RoboDK station: Yuchen_2024.rdk

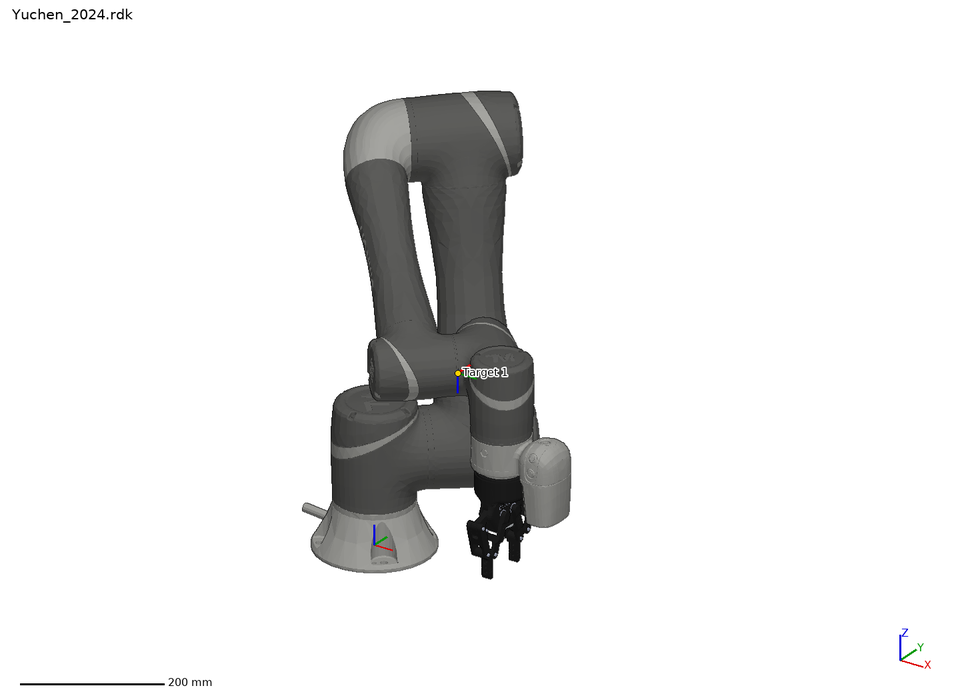
[picture v0: the station drawn from its stored meshes, robots at their saved joint values, targets as dots, program paths as lines]
Station Yuchen_2023 (saved by RoboDK 5.5.3). Poses are relative to the parent item; angles as X-Y-Z fixed-axis rotations.
  - frame Omron TM5-900 Base at (0, 0, 0) mm
    - robot Omron TM5-900: 6 axes, payload 4 kg, reach 900 mm, repeatability 0.1 mm, weight 30 kg
        modified DH rows (alpha deg, a mm, theta deg, d mm): 0, 0, 0, 145.2; 90, 0, 90, 0; 0, 429, 0, 0; 0, 411, -90, 122.3; -90, 0, 0, 106.5; 90, 0, 180, 114.15
        joint limits [-270, -180, -155, -180, -180, -270] to [270, 180, 155, 180, 180, 270]; home [0, 0, 90, -90, 90, 0]; saved at [134.48, 19.77, -133.5, 23.17, -90.14, -45.91]
      - tool RobotiQ 2F-85 Gripper (Closed), TCP at (0, 0, 130) mm, size 134.4 x 75 x 157.6 mm
    - frame Frame 2 at (241, -142.19, 389.18) mm, rotated rx -179.52 ry -0.29 rz 90.39 deg
      - target Target 1 (Cartesian target) at (0, 0, 0) mm; joints [123.542, 38.198, -125.271, -2.927, -90, -56.458] of Omron TM5-900
  - Python program Reading_CaseStudy (listed below)
  - Python program 20240725_OPT (listed below)

--- Python program Reading_CaseStudy ---
# PS C:\Users\Tesisti> python -m venv hrcreading
# PS C:\Users\Tesisti> .\hrcreading\Scripts\activate
# (hrcreading) PS C:\Users\Tesisti> C:/Python310/python.exe c:/Users/Tesisti/AppData/Local/Temp/Reading_CaseStudy_3.py

# import os
# os.environ['OPENAI_API_KEY'] ='sk-proj-5TX9ug0B6qDGBHHPTzqzT3BlbkFJDqqZnPh7HjYkSIwuRGDw'

# sys.path.append(yolov7_path)
# print("sys.path:", sys.path)
import cv2
import torch
import pyttsx3
from datetime import datetime
import numpy as np
import requests
from IPython.display import display, Audio
import openai
import time
from PIL import Image, ImageTk
import pandas as pd
import matplotlib.pyplot as plt
import pygame
import os
from GUI import AssemblyGUI
import tkinter as tk
from playsound import playsound
import sys
import tkinter as tk
from tkinter import ttk, messagebox
import pygame
from PIL import Image, ImageTk
from playsound import playsound


# from ultralytics.yolo.utils.downloads import non_max_suppression, check_img_size, scale_coords
# from utils.general import non_max_suppression, check_img_size, scale_coords
# from utils.torch_utils import select_device



# ———————————————————————————————————————————————————————————— GUI design ————————————————————————————————————————————————————————————
def load_and_play(speech=None):
    try:
        playsound(speech)
    except Exception as e:
        print(f"Error playing {speech}: {e}")

def pause_audio():
    pygame.mixer.music.pause()

def set_volume(value):
    volume_level = float(value) / 100
    pygame.mixer.music.set_volume(volume_level)

def change_voice(selected_voice_type):
    voice_type = selected_voice_type
    load_and_play()

def create_gui():
    root.title("Assembly Monitoring System")
    root.geometry("1200x800")  # Adjust window size

    # Frames for different sections
    left_column = tk.Frame(self.root, width=800, bg='white')
    right_column = tk.Frame(self.root, width=400, bg='light gray')
    left_column.pack(side='left', fill='both', expand=True)
    right_column.pack(side='right', fill='both', expand=True)

    # Sub-frames within the left frame
    image_display_frame = tk.Frame(left_column, width=800)
    label_description_0 = tk.Label(image_display_frame, text="Multi-form Instructions", font=('Arial', 16, 'bold'))
    label_description_0.pack(pady=(20, 0))
    image_display_frame.pack(side="top", fill="both", expand=True)
    command_frame = tk.Frame(left_column, width=400)
    command_frame.pack(side="top", fill="both", expand=False)

    # Sub-frames for each image and its description
    left_image_frame = tk.Frame(image_display_frame, width=400)
    right_image_frame = tk.Frame(image_display_frame, width=400)
    left_image_frame.pack(side="left", fill="both", expand=True)
    right_image_frame.pack(side="right", fill="both", expand=True)

    # Labels and images in the left image frame
    label_description_1 = tk.Label(left_image_frame, text="Component", font=('Arial', 14))
    canvas_com = tk.Canvas(left_image_frame, bg="gray", height=80, width=80)
    label_operation_1 = tk.Label(left_image_frame, text="Operation", font=('Arial', 14))
    canvas_ope = tk.Canvas(left_image_frame, bg="gray", height=80, width=80)
    label_description_1.pack(pady=(20, 0))
    canvas_com.pack(pady=(5, 5), fill="both", expand=True)
    label_operation_1.pack(pady=(5, 0))
    canvas_ope.pack(pady=(5, 20), fill="both", expand=True)

    # Labels and images in the right image frame
    label_description_2 = tk.Label(right_image_frame, text="Tool", font=('Arial', 14))
    canvas_too = tk.Canvas(right_image_frame, bg="gray", height=80, width=80)
    label_operation_2 = tk.Label(right_image_frame, text="Assembly Result", font=('Arial', 14))
    canvas_res = tk.Canvas(right_image_frame, bg="gray", height=80, width=80)
    label_description_2.pack(pady=(20, 0))
    canvas_too.pack(pady=(5, 5), fill="both", expand=True)
    label_operation_2.pack(pady=(5, 0))
    canvas_res.pack(pady=(5, 20), fill="both", expand=True)

    # Text box for instructions
    text_frame = tk.Frame(left_column, width=400)
    text_frame.pack(side="top", fill="both", expand=False, pady=(0, 0))
    text_instruction = tk.Text(text_frame, height=10, width=80)
    text_instruction.pack(pady=(5, 5), padx=0)

    # Main command frame for holding all control elements
    command_frame = tk.Frame(left_column, bg='white')
    command_frame.pack(fill="x")

    # Controls frame for holding buttons and sliders horizontally
    controls_frame = tk.Frame(command_frame)
    controls_frame.pack(fill="x", expand=True)

    # Buttons and controls in the command frame
    play_button = tk.Button(controls_frame, text="Play Instructions", font=('Arial', 12), command=load_and_play(speech=None))
    pause_button = tk.Button(controls_frame, text="Pause Instructions", font=('Arial', 12), command=pause_audio())
    volume_control = tk.Scale(controls_frame, from_=0, to=100, orient="horizontal", label="Volume", font=('Arial', 12), command=set_volume)
    volume_control.set(50)  # Default volume set to 50%
    sound_type = ttk.Combobox(controls_frame, values=["Male", "Female"], font=('Arial', 12), state="readonly")
    sound_type.set("Male")  # Default sound type
    play_button.grid(row=0, column=0, padx=10, pady=10, sticky="ew")
    pause_button.grid(row=0, column=1, padx=10, pady=10, sticky="ew")
    volume_control.grid(row=0, column=2, padx=10, pady=10, sticky="ew")
    sound_type.grid(row=0, column=3, padx=10, pady=10, sticky="ew")

    # Right column single image frame
    realtime_image_frame = tk.Frame(right_column, width=400, bg='light blue')
    realtime_image_frame.pack(side="top", fill="both", expand=True)
    label_description_3 = tk.Label(realtime_image_frame, text="Actual Statu", font=('Arial', 16, 'bold'), bg='light blue')
    label_description_3.pack(pady=(20, 0))

    # Image and label in the right column
    label_description_realtime = tk.Label(realtime_image_frame, text="Real-time Image", font=('Arial', 14), bg='light blue')
    realtime_canvas = tk.Canvas(realtime_image_frame, bg="gray", height=300, width=450)
    label_description_realtime.pack(pady=(20, 0))
    realtime_canvas.pack(pady=(5, 5), fill="none", expand=False)

    # Text box for assembly progress
    progress_frame = tk.Frame(right_column, width=400, bg='light blue')
    progress_frame.pack(side="top", fill="both", expand=False, pady=(0, 0))
    progress_label = tk.Label(progress_frame, text="Assembly Status", font=('Arial', 14), bg='light blue')
    progress_label.pack()
    progress_text = tk.Text(progress_frame, height=15, width=56)
    progress_text.pack(pady=(5, 20), padx=20)

    # Button frame at the bottom of right_column
    button_frame = tk.Frame(right_column, bg='light blue')
    button_frame.pack(side='bottom', fill='x', expand=False)
    exit_button = tk.Button(button_frame, text="Exit", font=('Arial', 12), command=root.destroy, width=10)
    error_button = tk.Button(button_frame, text="Report Error", font=('Arial', 12), command=lambda: messagebox.showerror("Error", "System Error Reported"), width=20)
    exit_button.pack(side="left", padx=35, pady=25)
    error_button.pack(side="right", padx=35, pady=25)




# ———————————————————————————————————————————————————————————— Data and model Setting ————————————————————————————————————————————————————————————
# YOLOv7
# loading the pre-trained YOLOv7 model
yolov7_path = 'C:/Users/Tesisti/Desktop/Yuchen 2023-2026/06 GPT+YOLOV7/yolov7'
weights_path = 'C:/Users/Tesisti/Desktop/Yuchen 2023-2026/06 GPT+YOLOV7/yolov7/best.pt'
device = torch.device('cuda' if torch.cuda.is_available() else 'cpu')
model = torch.hub.load(yolov7_path, 'custom', weights_path, source='local').to(device)
model.eval() # 确保模型处于评估模式
yolov7_label_order = ['Allen key', 'Hex cap screw (big)', 'Drive shaft companion flange', 'Nuts', 'Pump housing', 'S12', 'S6', 'S9', 'Washers', 'Wrench size 13']

# Assembly data loading
assembly_tasks_path = 'C:/Users/Tesisti/Desktop/Yuchen 2023-2026/06 GPT+YOLOV7/assembly_tasks.xlsx'
assembly_tasks_df = pd.read_excel(assembly_tasks_path)
index_total = assembly_tasks_df.dropna(how='all').shape[0] - 1

steps_classes = assembly_tasks_df['step'].dropna().to_dict()
components_classes = assembly_tasks_df['components'].dropna().to_dict()
tools_classes = assembly_tasks_df['tools'].dropna().to_dict()
operations_classes = assembly_tasks_df['operations'].dropna().to_dict()
time_classes = assembly_tasks_df['time'].dropna().to_dict()
lastorder_classes = assembly_tasks_df['lastorder'].dropna().to_dict()
print(steps_classes)
print(components_classes)
print(tools_classes)

# Error information
error_templates_path = 'C:/Users/Tesisti/Desktop/Yuchen 2023-2026/06 GPT+YOLOV7/error_templates.xlsx'
error_templates_df = pd.read_excel(error_templates_path)
error_templates = dict(zip(error_templates_df['error_type'], error_templates_df['template']))
print(error_templates)



# ———————————————————————————————————————————————————————————— Image Capture and Process ————————————————————————————————————————————————————————————
# Image display
def show_image(frame):
    try:
        frame_rgb = cv2.cvtColor(frame, cv2.COLOR_BGR2RGB)
        plt.imshow(frame_rgb)
        plt.axis('off')
        timestamp = datetime.now().strftime("%Y%m%d%H%M%S")
        plt.title(f'Image_{timestamp}')
        plt.show()  # Ensure the image is displayed when the function is called
    except Exception as e:
        print(f"Failed to display image: {e}")

# Image preprocessing
def preprocess_image(frame):
    try:
        img = cv2.cvtColor(frame, cv2.COLOR_BGR2RGB)
        img = img.astype(np.float32) / 255.0
        img = np.transpose(img, (2, 0, 1))
        img = np.expand_dims(img, 0)
        img = torch.from_numpy(img).float()
        return img
    except Exception as e:
        print(f"Error during image preprocessing: {e}")
        return None

# Image preprocessing cancel
def postprocess_image(tensor):
    if isinstance(tensor, torch.Tensor):
        tensor = tensor.cpu()
        image_np = tensor.numpy()
        image_np = image_np[0]
        if image_np.shape[0] < image_np.shape[2]:
            image_np = image_np.transpose(1, 2, 0)
        if image_np.max() <= 1.0:
            image_np = (image_np * 255).astype(np.uint8)
        return image_np
    else:
        print("传入的数据不是 torch.Tensor 类型")
        return None

# Image capturing
def capture_image():
    cap = cv2.VideoCapture(0)
    ret, frame = cap.read()
    cap.release()
    if ret:
        # show_image(frame)
        img = preprocess_image(frame)
        return img
    else:
        return None


# ———————————————————————————————————————————————————————————— YOLOv7 Detection and classification ————————————————————————————————————————————————————————————
# Image YOLOv7 detection
def detect_items(image):
    frame = image.squeeze().numpy().transpose(1, 2, 0) * 255  # 转换图像为适合显示的格式
    frame = frame.astype(np.uint8)

    with torch.no_grad():
        predictions = model(image)  # 使用模型进行预测
        predictions = predictions[0] if isinstance(predictions, tuple) else predictions
        predictions = non_max_suppression(predictions, conf_thres=0.6, iou_thres=0.45)

    detected_items = []  # 初始化检测到的物体列表

    # 检查predictions是否存在且不为空
    if predictions is not None and len(predictions) > 0 and len(predictions[0]) > 0:
        detected_items = predictions[0]  # 提取检测到的物体
        print(f"YOLOv7 detections found: {len(detected_items)}")  # 打印检测到的物体数量
    else:
        print("No detections found.")

    return detected_items

# detected items classification
def classify_detections(detected):
    classified_items = {
        'components': [],
        'tools': [],
        'steps': []
    }
    for detection in detected:
        x1, y1, x2, y2, conf, cls = detection[:6]
        if conf > 0.5:
            label = yolov7_label_order[int(cls)]
            print('label:' + label)
            if any(label == step for step in steps_classes.values()):
                classified_items['steps'].append(label)
            if any(label in component for component in components_classes.values()):
                classified_items['components'].append(label)
            if any(label in tool for tool in tools_classes.values()):
                classified_items['tools'].append(label)
    return classified_items



# ———————————————————————————————————————————————————————————— Annotate by Error ————————————————————————————————————————————————————————————
# Error validation and handle
def error_validation(classified, step_details, operator_name, location, item_type, task):
    details = {
        'now': datetime.now().strftime("%Y-%m-%d %H:%M"),
        'operator_name': operator_name,
        'location': location,
        'expected': step_details[item_type],
        'actual': classified[item_type],
        'step': step_details['step'],
        'task': task
    }

    error_result = {
        'type': item_type,
        'specific': details['actual'],
        'result': True
    }

    if set(details['actual']).issubset(set(details['expected'])):
        error_result['result'] = True
        error_log = None
    else:
        error_result['result'] = False
        error_log = error_templates[item_type].format(**details)  # Ensure error_templates is defined with proper templates.

    errorLog_dir = "C:/Users/Tesisti/Desktop/Yuchen 2023-2026/06 GPT+YOLOV7/Results_ErrorLog"
    current_time = datetime.now().strftime("%Y-%m-%d_%H-%M-%S")
    errorLog_filename = f"{errorLog_dir}/text{current_time}.txt"
    with open(errorLog_filename, "w") as text_file:
        text_file.write(error_log)
    print(f"Error log saved.")

    return error_result, error_log

# Label with different colors according to different situation
def annotate_image_with_labels(image, detected_items, classified_items, item_type, error_result):
    # Define colors for different scenarios
    correct_color = (0, 255, 0)  # Green for "True"
    wrong_color = (255, 0, 0)    # Red for "False"
    neutral_color = (128, 128, 128)  # Gray for other categories

    # Process the image once
    processed_image = postprocess_image(image)

    for detection in detected_items:
        x1, y1, x2, y2, conf, cls = detection[:6]
        detection_label = yolov7_label_order[int(cls)]  # Convert class ID to readable label

        # Determine the color based on classification and result
        if detection_label in classified_items[item_type]:
            color = correct_color if error_result['result'] else wrong_color
        else:
            color = neutral_color

        # Draw rectangle and label on the same processed image
        cv2.rectangle(processed_image, (int(x1), int(y1)), (int(x2), int(y2)), color, 2)
        cv2.putText(processed_image, detection_label, (int(x1), int(y1) - 10), cv2.FONT_HERSHEY_SIMPLEX, 0.5, color, 2)

    # Save and optionally display the annotated image
    timestamp = datetime.now().strftime("%Y%m%d%H%M%S")
    annotated_image_path = f'./Results_Image/annotated_{item_type}_{timestamp}.jpg'
    cv2.imwrite(annotated_image_path, processed_image)
    print(f"Annotated image saved.")

    return processed_image



# ———————————————————————————————————————————————————————————— GPT promt and speech ————————————————————————————————————————————————————————————
# Load gpt prompt
def generate_prompt(step_details, error_description):
    gpt_prompt_path = 'C:/Users/Tesisti/Desktop/Yuchen 2023-2026/06 GPT+YOLOV7/gpt_prompt.xlsx'
    gpt_prompt_df = pd.read_excel(gpt_prompt_path)
    prompt_template = gpt_prompt_df['prompt'].iloc[0]
    prompt = prompt_template.format(step_details=step_details, error_description=error_description)
    return prompt

def GPT_TTS(prompt):
    # Check GPT API key
    api_key = os.getenv('OPENAI_API_KEY')
    if not api_key:
        raise ValueError("API key is not set. Please ensure the 'OPENAI_API_KEY' environment variable is defined.")

    # Step1: Text generation
    response = openai.chat.completions.create(
        model="gpt-4o",
        messages=[{"role": "user", "content": prompt}]
    )
    text = response.choices[0].message.content.strip()
    # print("Generated text:", text)

    # Text result save
    results_text_dir = "C:/Users/Tesisti/Desktop/Yuchen 2023-2024/06 GPT+YOLOV7/Results_Text"
    current_time = datetime.now().strftime("%Y-%m-%d_%H-%M-%S")
    text_filename = f"{results_text_dir}/text{current_time}.txt"
    with open(text_filename, "w") as text_file:
        text_file.write(text)
    print(f"Results text saved.")

    # Step2: Speech generation
    headers = {
        'Authorization': f'Bearer {api_key}',
        'Content-Type': 'application/json',
    }
    data = {
        "model": "tts-1",
        "input": text,
        "voice": "alloy"
    }
    response = requests.post('https://api.openai.com/v1/audio/speech', headers=headers, json=data)
    if response.status_code == 200:
        results_speech_dir = "C:/Users/Tesisti/Desktop/Yuchen 2023-2026/06 GPT+YOLOV7/Results_Speech"
        speech_filename = f"{results_speech_dir}/speech{current_time}.mp3"
        with open(speech_filename, 'wb') as file:
            file.write(response.content)
        print("Error instruction speech saved.")
        # display(Audio(speech_filename, autoplay=True))
    else:
        print("Failed to generate speech:", response.status_code, response.text)
    return speech_filename

# Text to speech
def text_to_speech(text):
    timestamp = datetime.now().strftime("%Y%m%d%H%M%S")
    voice_path = f'C:/Users/Tesisti/Desktop/Yuchen 2023-2026/06 GPT+YOLOV7/TTS_Speech/voice_{timestamp}.mp3'
    try:
        engine = pyttsx3.init()
        rate = engine.getProperty('rate')  # Obatain current speed
        engine.setProperty('rate', rate - 80)  # Modify speed
        volume = engine.getProperty('volume')  # Obatain current volume
        engine.setProperty('volume', volume + 0.25)  # Modify volume
        voices = engine.getProperty('voices')  # Obatain aviable voice
        engine.setProperty('voice', voices[0].id)  # Modify voice（0-male，1-female）
        engine.say(text)
        engine.save_to_file(text, voice_path)
        engine.runAndWait()
        return voice_path
    except Exception as e:
        print(f"Error with text-to-speech: {e}")
        return None
        # print(text)

def play_audio(filename):
    # pygame.mixer.init()
    pygame.mixer.music.load(filename)
    pygame.mixer.music.play()
    while pygame.mixer.music.get_busy():
        pygame.time.Clock().tick(10)



# ———————————————————————————————————————————————————————————— GUI Update ————————————————————————————————————————————————————————————
# 更新四大块图像的显示：canvas_com，canvas_ope，canvas_too，canvas_res
def update_gui_4image(gui, step):
    base_path = 'C:/Users/Tesisti/Desktop/Yuchen 2023-2026/06 GPT+YOLOV7/CS_CIRP2024/'

    # 构建每个图像的完整路径和对应的画布
    image_paths = {
        'component': f'{base_path}component/step{step}_com.png',
        'tool': f'{base_path}tool/step{step}_too.png',
        'operation': f'{base_path}operation/step{step}_ope.png',
        'result': f'{base_path}result/step{step}_res.png'
    }

    canvases = {
        'component': gui.canvas_com,
        'tool': gui.canvas_too,
        'operation': gui.canvas_ope,
        'result': gui.canvas_res
    }

    # 循环检查每个图像路径并更新相应的画布
    for key, path in image_paths.items():
        canvas = canvases[key]
        if os.path.exists(path):
            img = Image.open(path)
            img = img.resize((canvas.winfo_width(), canvas.winfo_height()), Image.Resampling.LANCZOS) #Image.ANTIALIAS
            img = ImageTk.PhotoImage(img)
            canvas.image = img
            canvas.create_image(0, 0, anchor='nw', image=img)
        else:
            canvas.delete("all")



# ———————————————————————————————————————————————————————————— Main Function ————————————————————————————————————————————————————————————
# main
def main():
    GUI = AssemblyGUI()
    operator_name = input("Please enter the operator's name: ")
    location = "Assembly Line 3, Workstation 7"

    pygame.mixer.init()
    # GUI.create_gui()
    # update_gui()

    for index in range(index_total):
        # Obtain all the information for this step
        step_details = {
            'components': components_classes[index],
            'tools': tools_classes[index],
            'operations': operations_classes[index],
            'time': time_classes[index],
            'step': steps_classes[index],
            'steps': steps_classes[index]
        }
        GUI.progress_text.delete('1.0', tk.END) # 清空GUI的process框中的所有文字内容
        step_number = int(step_details['step'][1:])
        update_gui_4image(GUI, step_number) # 根据当下步骤更新GUI左上角的四张图
        # print(step_details)

        for item_type in ['components', 'tools', 'steps']:
            text = f"Start assembly step{index+1}.{item_type}."
            GUI.progress_text.insert(tk.END, text) # 更新GUI的process框中的文字内容
            GUI.root.update_idletasks()
            if step_details[item_type] != "None":
                retry = True
                retry_count = 0
                while retry and retry_count < 3:
                    timestamp = datetime.now().strftime("%Y%m%d%H%M%S")
                    file_name = f"{item_type}_{timestamp}.mp4"
                    if item_type in ['components', 'tools']:
                        Task = f"Please prepare the following {item_type}: {step_details[item_type]}."
                        sleep_time = 6
                    else:
                        Task = f"Please follow the instructions to complete the step: {step_details['operations']}."
                        sleep_time = step_details['time']

                    GUI.text_instruction.delete('1.0', tk.END)
                    GUI.text_instruction.insert(tk.END, Task) # 更新GUI的instruction框中的文字内容
                    GUI.root.update_idletasks()
                    voice = text_to_speech(Task)
                    print(voice)
                    GUI.load_and_play(voice) # 更新GUI的播放button的command
                    GUI.root.update_idletasks()
                    # play_audio(voice)

                    time.sleep(sleep_time)

                    image = capture_image()
                    image_np = postprocess_image(image) # 把图像从tensor格式转换到numpy
                    image_pil = Image.fromarray(image_np)  # 把图像从numpy格式转换到pil
                    photo_image = ImageTk.PhotoImage(image_pil)
                    GUI.realtime_canvas.image = photo_image
                    GUI.realtime_canvas.create_image(0, 0, anchor='nw', image=photo_image) # 更新GUI的realtime image框中的图片
                    GUI.root.update_idletasks()

                    detected_items = detect_items(image)
                    text = f"\nDetected: {detected_items}."
                    GUI.progress_text.insert(tk.END, text) # 更新GUI的process框中的文字内容
                    GUI.root.update_idletasks()
                    # print(detected_items)
                    classified_items = classify_detections(detected_items)
                    # print(classified_items)
                    error_result, error_log = error_validation(classified_items, step_details, operator_name, location, item_type, Task)
                    # print(error_log)
                    text = f"\nError Log: {error_log}."
                    GUI.progress_text.insert(tk.END, text) # 更新GUI的process框中的文字内容

                    image = annotate_image_with_labels(image, detected_items, classified_items, item_type, error_result)
                    GUI.realtime_canvas.image = image
                    GUI.realtime_canvas.create_image(0, 0, anchor='nw', image=image) # 更新GUI的realtime image框中的图片

                    if error_result['result'] == False:
                        if retry_count < 2:
                            prompt = generate_prompt(step_details, error_log)
                            speech_filename = GPT_TTS(prompt)
                            play_audio(speech_filename)
                            text = f"\nRedo step{index+1}.{item_type}"
                            GUI.progress_text.insert(tk.END, text) # 更新GUI的process框中的文字内容
                            retry_count += 1
                        else:
                            text = f"\nFailed to correct the error after 2 attempts."
                            GUI.progress_text.insert(tk.END, text) # 更新GUI的process框中的文字内容
                            retry = False
                    else:
                        text = f"\nYou did it correctly. Now let's proceed to the next step."
                        voice = text_to_speech(text)
                        play_audio(voice)
                        GUI.progress_text.insert(tk.END, text) # 更新GUI的process框中的文字内容
                        text = f"\nEnd step{index+1}.{item_type}"
                        GUI.progress_text.insert(tk.END, text) # 更新GUI的process框中的文字内容
                        retry = False

    GUI.run()

if __name__ == '__main__':
    main()

--- Python program 20240725_OPT ---
# 建立虚拟环境，环境名：hrcreading
# PS C:\Users\Tesisti> python -m venv hrcreading
# PS C:\Users\Tesisti> .\hrcreading\Scripts\activate
# (hrcreading) PS C:\Users\Tesisti> C:/Python310/python.exe c:/Users/Tesisti/AppData/Local/Temp/Reading_CaseStudy_3.py

# 在环境中写入GPT的API
# $env:OPENAI_API_KEY = "sk-proj-5TX9ug0B6qDGBHHPTzqzT3BlbkFJDqqZnPh7HjYkSIwuRGDw"
# $env:OPENAI_API_KEY

import os
import sys
import time
from datetime import datetime
import cv2
import torch
import numpy as np
import pandas as pd
import tkinter as tk
from tkinter import ttk, messagebox
from PIL import Image, ImageTk
import matplotlib
matplotlib.use('Agg')  # 在导入pyplot之前设置backend
import matplotlib.pyplot as plt
import pygame
from playsound import playsound
import pyttsx3
import requests
import openai
from IPython.display import display, Audio
from tkinter import simpledialog
import torch.nn.functional as F
import torch
from ultralytics import YOLO
import yolov7
import torchvision
import threading

# 配置管理
CONFIG = {
    'yolov7_path': 'C:/Users/Tesisti/Desktop/Yuchen 2023-2026/06 GPT+YOLOV7/yolov7',
    'weights_path': 'C:/Users/Tesisti/Desktop/Yuchen 2023-2026/06 GPT+YOLOV7/yolov7/best.pt',
    'assembly_tasks_path': 'C:/Users/Tesisti/Desktop/Yuchen 2023-2026/06 GPT+YOLOV7/assembly_tasks.xlsx',
    'error_templates_path': 'C:/Users/Tesisti/Desktop/Yuchen 2023-2026/06 GPT+YOLOV7/error_templates.xlsx',
    'gpt_prompt_path': 'C:/Users/Tesisti/Desktop/Yuchen 2023-2026/06 GPT+YOLOV7/gpt_prompt.xlsx',
    'instruction_path': 'C:/Users/Tesisti/Desktop/Yuchen 2023-2026/06 GPT+YOLOV7/CS_CIRP2024/',
    'results_image_dir': 'C:/Users/Tesisti/Desktop/Yuchen 2023-2026/06 GPT+YOLOV7/Results_Image',
    'results_text_dir': 'C:/Users/Tesisti/Desktop/Yuchen 2023-2026/06 GPT+YOLOV7/Results_Text',
    'results_errorlog_dir': 'C:/Users/Tesisti/Desktop/Yuchen 2023-2026/06 GPT+YOLOV7/Results_ErrorLog',
    'results_speech_dir': 'C:/Users/Tesisti/Desktop/Yuchen 2023-2026/06 GPT+YOLOV7/Results_Speech',
    'TTS_speech_dir': 'C:/Users/Tesisti/Desktop/Yuchen 2023-2026/06 GPT+YOLOV7/TTS_Speech',
    'tts_voice': 'alloy'
}

class AssemblyMonitoringSystem():
    def __init__(self, window): # 全系统初始化
        self.window = window
        self.initialize_gui()
        self.operator_name = self.get_operator_name()
        self.load_data()
        self.initialize_model()
        pygame.mixer.init()
        self.current_audio_file = None
        self.window.protocol("WM_DELETE_WINDOW", self.on_closing)
        self.yolov7_label_order = ['Allen key', 'Hex cap screw (big)', 'Drive shaft companion flange', 'Nuts', 'Pump housing', 'S12', 'S6', 'S9', 'Washers', 'Wrench size 13']

    def load_data(self): # 加载数据：1)装配任务，2)错误模板，3)GPT prompt模板.
        self.assembly_tasks_df = pd.read_excel(CONFIG['assembly_tasks_path'])
        self.error_templates_df = pd.read_excel(CONFIG['error_templates_path'])
        self.gpt_prompt_df = pd.read_excel(CONFIG['gpt_prompt_path'])
        self.error_templates = dict(zip(self.error_templates_df['error_type'], self.error_templates_df['template']))

    def initialize_model(self): # 初始化 YOLOv7 模型
        # self.device = torch.device('cuda' if torch.cuda.is_available() else 'cpu')
        self.device = torch.device('cpu')
        self.model = torch.hub.load(CONFIG['yolov7_path'], 'custom', CONFIG['weights_path'], source='local').to(self.device)
        self.model.eval()

    def get_operator_name(self): # 获取操作者名字
        name = simpledialog.askstring("Input", "Please enter the operator's name:", parent=self.window)
        return name if name else "Unknown Operator"

    def initialize_gui(self): # GUI初始化
        # 创建 GUI 元素
        self.window.title("Assembly Monitoring System")
        self.window.geometry("1400x900")
        pygame.mixer.init()

        # 创建左右列
        self.left_column = tk.Frame(self.window, width=800, bg='white')
        self.right_column = tk.Frame(self.window, width=600, bg='light gray')
        self.left_column.pack(side='left', fill='both', expand=True)
        self.right_column.pack(side='right', fill='both', expand=True)

        # 创建左列的子框架
        self.image_display_frame = tk.Frame(self.left_column, width=800)
        label_description_0 = tk.Label(self.image_display_frame, text="Multi-form Instructions", font=('Arial', 16, 'bold'))
        label_description_0.pack(pady=(20, 0))
        self.image_display_frame.pack(side="top", fill="both", expand=True)
        self.command_frame = tk.Frame(self.left_column, width=400)
        self.command_frame.pack(side="top", fill="both", expand=False)

        # 创建左列图像显示区域
        self.left_image_frame = tk.Frame(self.image_display_frame, width=400)
        self.right_image_frame = tk.Frame(self.image_display_frame, width=400)
        self.left_image_frame.pack(side="left", fill="both", expand=True)
        self.right_image_frame.pack(side="right", fill="both", expand=True)

        self.canvas_com = tk.Canvas(self.left_image_frame, bg="gray", height=80, width=80)
        self.label_description_1 = tk.Label(self.left_image_frame, text="Component", font=('Arial', 14))
        self.label_description_1.pack(pady=(20, 0))
        self.canvas_com.pack(pady=(5, 5), fill="both", expand=True)

        self.canvas_ope = tk.Canvas(self.left_image_frame, bg="gray", height=80, width=80)
        self.label_operation_1 = tk.Label(self.left_image_frame, text="Operation", font=('Arial', 14))
        self.label_operation_1.pack(pady=(5, 0))
        self.canvas_ope.pack(pady=(5, 20), fill="both", expand=True)

        self.canvas_too = tk.Canvas(self.right_image_frame, bg="gray", height=80, width=80)
        self.label_description_2 = tk.Label(self.right_image_frame, text="Tool", font=('Arial', 14))
        self.label_description_2.pack(pady=(20, 0))
        self.canvas_too.pack(pady=(5, 5), fill="both", expand=True)

        self.canvas_res = tk.Canvas(self.right_image_frame, bg="gray", height=80, width=80)
        self.label_operation_2 = tk.Label(self.right_image_frame, text="Assembly Result", font=('Arial', 14))
        self.label_operation_2.pack(pady=(5, 0))
        self.canvas_res.pack(pady=(5, 20), fill="both", expand=True)

        self.text_frame = tk.Frame(self.left_column, width=400)
        self.text_frame.pack(side="top", fill="both", expand=False, pady=(0, 0))
        self.text_instruction = tk.Text(self.text_frame, height=10, width=80)
        self.text_instruction.config(font=('Arial', 12))
        self.text_instruction.pack(pady=(5, 5), padx=0)

        self.command_frame = tk.Frame(self.left_column, bg='white')
        self.command_frame.pack(fill="x")

        self.controls_frame = tk.Frame(self.command_frame)
        self.controls_frame.pack(fill="x", expand=True)

        self.play_button = tk.Button(self.controls_frame, text="Play Instructions", font=('Arial', 12), command=lambda: self.audio_control('load_and_play'))
        self.pause_button = tk.Button(self.controls_frame, text="Pause Instructions", font=('Arial', 12), command=lambda: self.audio_control('pause'))
        self.volume_control = tk.Scale(self.controls_frame, from_=0, to=100, orient="horizontal", label="Volume", font=('Arial', 12), command=lambda x: self.audio_control('set_volume', x))
        self.sound_type = ttk.Combobox(self.controls_frame, values=["alloy", "echo", "fable", "onyx", "nova", "shimmer"], font=('Arial', 12), state="readonly")
        self.sound_type.set("alloy")
        self.play_button.grid(row=0, column=0, padx=20, pady=10, sticky="ew")
        self.pause_button.grid(row=0, column=1, padx=20, pady=10, sticky="ew")
        self.volume_control.grid(row=0, column=2, padx=20, pady=10, sticky="ew")
        self.sound_type.grid(row=0, column=3, padx=20, pady=10, sticky="ew")

        # 创建右列的子框架
        self.realtime_image_frame = tk.Frame(self.right_column, width=400, bg='light blue')
        self.realtime_image_frame.pack(side="top", fill="both", expand=True)
        label_description_3 = tk.Label(self.realtime_image_frame, text="Actual Status", font=('Arial', 16, 'bold'), bg='light blue')
        label_description_3.pack(pady=(20, 0))

        label_description_realtime = tk.Label(self.realtime_image_frame, text="Real-time Image", font=('Arial', 14), bg='light blue')
        self.realtime_canvas = tk.Canvas(self.realtime_image_frame, bg="gray", height=400, width=550)
        label_description_realtime.pack(pady=(20, 0))
        self.realtime_canvas.pack(pady=(5, 5), fill="none", expand=False)

        self.progress_frame = tk.Frame(self.right_column, width=400, bg='light blue')
        self.progress_frame.pack(side="top", fill="both", expand=False, pady=(0, 0))
        progress_label = tk.Label(self.progress_frame, text="Assembly Progress", font=('Arial', 14), bg='light blue')
        progress_label.pack()
        self.progress_text = tk.Text(self.progress_frame, height=13, width=56)
        self.progress_text.config(font=('Arial', 12))
        self.progress_text.pack(pady=(5, 20), padx=20)

        self.button_frame = tk.Frame(self.right_column, bg='light blue', height=40)
        self.button_frame.pack(side='bottom', fill='x', expand=False)
        self.exit_button = tk.Button(self.button_frame, text="Exit", font=('Arial', 12), command=self.window.destroy, width=10)
        self.error_button = tk.Button(self.button_frame, text="Report Error", font=('Arial', 12), command=lambda: messagebox.showerror("Error", "System Error Reported"), width=20)
        self.exit_button.pack(side="left", padx=35, pady=25)
        self.error_button.pack(side="right", padx=35, pady=25)

    def play_audio(self, filename): # 播放音频
        if filename and os.path.exists(filename):
            try:
                self.current_audio_file = filename
                pygame.mixer.music.load(filename)
                pygame.mixer.music.play()
                while pygame.mixer.music.get_busy():
                    pygame.time.Clock().tick(10)
            except Exception as e:
                print(f"Error playing audio: {e}")
        else:
            print(f"Audio file not found: {filename}")

    def update_gui_4image(self, step): # 更新四个图像显示区域
        image_paths = {
            'component': f'{CONFIG["instruction_path"]}/component/step{step}_com.png',
            'tool': f'{CONFIG["instruction_path"]}/tool/step{step}_too.png',
            'operation': f'{CONFIG["instruction_path"]}/operation/step{step}_ope.png',
            'result': f'{CONFIG["instruction_path"]}/result/step{step}_res.png'
        }
        canvases = {
            'component': self.canvas_com,
            'tool': self.canvas_too,
            'operation': self.canvas_ope,
            'result': self.canvas_res
        }
        for key, path in image_paths.items():
            canvas = canvases[key]
            if os.path.exists(path):
                img = Image.open(path)
                img = img.resize((canvas.winfo_width(), canvas.winfo_height()), Image.Resampling.LANCZOS)
                img = ImageTk.PhotoImage(img)
                canvas.image = img
                canvas.create_image(0, 0, anchor='nw', image=img)
            else:
                canvas.delete("all")
        self.window.update()

    def update_realtime_image(self, image): # 更新实时图像显示区域
        try:
            if isinstance(image, torch.Tensor):
                image = self.postprocess_image(image)

            if isinstance(image, np.ndarray):
                # 确保图像是 RGB 格式
                if image.shape[2] == 3:
                    image_rgb = cv2.cvtColor(image, cv2.COLOR_BGR2RGB)
                else:
                    image_rgb = image
                image_pil = Image.fromarray(image_rgb)
            elif isinstance(image, Image.Image):
                image_pil = image
            else:
                print(f"Unexpected image type: {type(image)}")
                return

            # 调整图像大小
            resized_image = image_pil.resize((self.realtime_canvas.winfo_width(), self.realtime_canvas.winfo_height()), Image.Resampling.LANCZOS)

            photo_image = ImageTk.PhotoImage(resized_image)

            self.realtime_canvas.delete("all")  # 清除旧的图像
            self.realtime_canvas.image = photo_image  # 保持对图像的引用
            self.realtime_canvas.create_image(0, 0, anchor='nw', image=photo_image)

            self.window.update()
        except Exception as e:
            print(f"Error updating realtime image: {e}")

    def update_instruction_text(self, text): # 更新指令显示的文字区域
        self.text_instruction.delete('1.0', tk.END)
        self.text_instruction.insert(tk.END, text)
        self.text_instruction.update()  # 强制更新
        self.window.update()  # 更新整个窗口

    def update_progress_text(self, text): # 更新进度显示的文字区域
        self.progress_text.insert(tk.END, text)

    def audio_control(self, action, value=None): # 控制音频（播放，暂停，调整音量）
        if action == 'load_and_play':
            if self.current_audio_file and os.path.exists(self.current_audio_file):
                try:
                    pygame.mixer.music.load(self.current_audio_file)
                    pygame.mixer.music.play()
                except Exception as e:
                    print(f"Error playing {self.current_audio_file}: {e}")
            else:
                print("No audio file available to play")
        elif action == 'pause':
            pygame.mixer.music.pause()
        elif action == 'set_volume':
            volume_level = float(value) / 100
            pygame.mixer.music.set_volume(volume_level)

    def capture_image(self): # 捕捉实时图像
        cap = cv2.VideoCapture(0)
        ret, frame = cap.read()
        cap.release()
        if ret:
            return frame  # 返回原始图像，不进行预处理
        else:
            print("Failed to capture image")
            return None

    def preprocess_image(self, frame):
        try:
            if frame is None:
                print("Input frame is None")
                return None
            img = cv2.cvtColor(frame, cv2.COLOR_BGR2RGB)
            img = img.astype(np.float32) / 255.0
            img = np.transpose(img, (2, 0, 1))
            img = np.expand_dims(img, 0)
            img = torch.from_numpy(img).float()
            return img
        except Exception as e:
            print(f"Error during image preprocessing: {e}")
            return None

    def postprocess_image(self, tensor): # 将模型输出的PyTorch张量转换回可以显示或进一步处理的NumPy数组
        if isinstance(tensor, torch.Tensor):
            tensor = tensor.cpu()
            image_np = tensor.numpy()
            image_np = image_np[0]
            if image_np.shape[0] < image_np.shape[2]:
                image_np = image_np.transpose(1, 2, 0)
            if image_np.max() <= 1.0:
                image_np = (image_np * 255).astype(np.uint8)
            return image_np
        elif isinstance(tensor, np.ndarray):
            return tensor  # 如果已经是numpy数组，直接返回
        else:
            print(f"Unexpected data type in postprocess_image: {type(tensor)}")
            return None

    def enhance_image(self, image): # 增强图像的亮度和饱和度
        # 转换到 HSV 色彩空间
        hsv = cv2.cvtColor(image, cv2.COLOR_BGR2HSV).astype("float32")
        (h, s, v) = cv2.split(hsv)

        # 增加亮度
        v = v * 1.4  # 增加 20% 的亮度
        v = np.clip(v, 0, 255)

        # 增加饱和度
        s = s * 1.3  # 增加 30% 的饱和度
        s = np.clip(s, 0, 255)

        # 合并通道
        hsv = cv2.merge([h, s, v])

        # 转换回 BGR 色彩空间
        enhanced_image = cv2.cvtColor(hsv.astype("uint8"), cv2.COLOR_HSV2BGR)

        return enhanced_image

    def detect_items(self, image): # YOLOv7检测
        print(f"Image shape: {image.shape}")
        print(f"Image dtype: {image.dtype}")
        print(f"Image device: {image.device}")
        print(f"Image max value: {image.max()}")
        print(f"Image min value: {image.min()}")

        if image is None:
            print("Input image is None")
            return []

        with torch.no_grad():
            predictions = self.model(image)  # 使用模型进行预测
            predictions = predictions[0] if isinstance(predictions, tuple) else predictions
            predictions = self.non_max_suppression(predictions, conf_thres=0.6, iou_thres=0.45)

        detected_items = []  # 初始化检测到的物体列表

        # 检查predictions是否存在且不为空
        if predictions is not None and len(predictions) > 0 and len(predictions[0]) > 0:
            detected_items = predictions[0].cpu().numpy()  # 提取检测到的物体并转换为numpy数组
            print(f"YOLOv7 detections found: {len(detected_items)}")  # 打印检测到的物体数量

            for det in detected_items:
                x1, y1, x2, y2, conf, cls = det
                print(f"Detected {self.yolov7_label_order[int(cls)]} with confidence {conf:.2f} at location [{x1:.1f}, {y1:.1f}, {x2:.1f}, {y2:.1f}]")
        else:
            print("No detections found.")

        return detected_items

    def non_max_suppression(self, prediction, conf_thres=0.25, iou_thres=0.7, classes=None, agnostic=False, multi_label=False, labels=()): # 去除冗余的检测框
        """Runs Non-Maximum Suppression (NMS) on inference results

        Returns:
            list of detections, on (n,6) tensor per image [xyxy, conf, cls]
        """

        nc = prediction.shape[2] - 5  # number of classes
        xc = prediction[..., 4] > conf_thres  # candidates

        # Settings
        min_wh, max_wh = 2, 4096  # (pixels) minimum and maximum box width and height
        max_det = 300  # maximum number of detections per image
        max_nms = 30000  # maximum number of boxes into torchvision.ops.nms()
        time_limit = 10.0  # seconds to quit after
        redundant = True  # require redundant detections
        multi_label &= nc > 1  # multiple labels per box (adds 0.5ms/img)
        merge = False  # use merge-NMS

        t = time.time()
        output = [torch.zeros((0, 6), device=prediction.device)] * prediction.shape[0]
        for xi, x in enumerate(prediction):  # image index, image inference
            # Apply constraints
            # x[((x[..., 2:4] < min_wh) | (x[..., 2:4] > max_wh)).any(1), 4] = 0  # width-height
            x = x[xc[xi]]  # confidence

            # Cat apriori labels if autolabelling
            if labels and len(labels[xi]):
                l = labels[xi]
                v = torch.zeros((len(l), nc + 5), device=x.device)
                v[:, :4] = l[:, 1:5]  # box
                v[:, 4] = 1.0  # conf
                v[range(len(l)), l[:, 0].long() + 5] = 1.0  # cls
                x = torch.cat((x, v), 0)

            # If none remain process next image
            if not x.shape[0]:
                continue

            # Compute conf
            if nc == 1:
                x[:, 5:] = x[:, 4:5] # for models with one class, cls_loss is 0 and cls_conf is always 0.5,
                                    # so there is no need to multiplicate.
            else:
                x[:, 5:] *= x[:, 4:5]  # conf = obj_conf * cls_conf

            # Box (center x, center y, width, height) to (x1, y1, x2, y2)
            box = self.xywh2xyxy(x[:, :4])

            # Detections matrix nx6 (xyxy, conf, cls)
            if multi_label:
                i, j = (x[:, 5:] > conf_thres).nonzero(as_tuple=False).T
                x = torch.cat((box[i], x[i, j + 5, None], j[:, None].float()), 1)
            else:  # best class only
                conf, j = x[:, 5:].max(1, keepdim=True)
                x = torch.cat((box, conf, j.float()), 1)[conf.view(-1) > conf_thres]

            # Filter by class
            if classes is not None:
                x = x[(x[:, 5:6] == torch.tensor(classes, device=x.device)).any(1)]

            # Apply finite constraint
            # if not torch.isfinite(x).all():
            #     x = x[torch.isfinite(x).all(1)]

            # Check shape
            n = x.shape[0]  # number of boxes
            if not n:  # no boxes
                continue
            elif n > max_nms:  # excess boxes
                x = x[x[:, 4].argsort(descending=True)[:max_nms]]  # sort by confidence

            # Batched NMS
            c = x[:, 5:6] * (0 if agnostic else max_wh)  # classes
            boxes, scores = x[:, :4] + c, x[:, 4]  # boxes (offset by class), scores
            i = torchvision.ops.nms(boxes, scores, iou_thres)  # NMS
            if i.shape[0] > max_det:  # limit detections
                i = i[:max_det]
            if merge and (1 < n < 3E3):  # Merge NMS (boxes merged using weighted mean)
                # update boxes as boxes(i,4) = weights(i,n) * boxes(n,4)
                iou = box_iou(boxes[i], boxes) > iou_thres  # iou matrix
                weights = iou * scores[None]  # box weights
                x[i, :4] = torch.mm(weights, x[:, :4]).float() / weights.sum(1, keepdim=True)  # merged boxes
                if redundant:
                    i = i[iou.sum(1) > 1]  # require redundancy

            output[xi] = x[i]
            if (time.time() - t) > time_limit:
                print(f'WARNING: NMS time limit {time_limit}s exceeded')
                break  # time limit exceeded

        return output

    def xywh2xyxy(self, x): # 坐标格式转换函数, 用于NMS
        # Convert nx4 boxes from [x, y, w, h] to [x1, y1, x2, y2] where xy1=top-left, xy2=bottom-right
        y = x.clone() if isinstance(x, torch.Tensor) else np.copy(x)
        y[:, 0] = x[:, 0] - x[:, 2] / 2  # top left x
        y[:, 1] = x[:, 1] - x[:, 3] / 2  # top left y
        y[:, 2] = x[:, 0] + x[:, 2] / 2  # bottom right x
        y[:, 3] = x[:, 1] + x[:, 3] / 2  # bottom right y
        return y

    def classify_detections(self, detected):  # 把YOLOv7模型检测出来的物体进行分类
        classified_items = {
            'components': [],
            'tools': [],
            'steps': []
        }

        for detection in detected:
            x1, y1, x2, y2, conf, cls = detection[:6]
            if conf > 0.5:
                detected_label = self.yolov7_label_order[int(cls)]
                print('Detected label:', detected_label)

                # 检查步骤
                if any(detected_label in step for step in self.steps_classes.values()):
                    classified_items['steps'].append(detected_label)
                    print(f'Matched to step: {detected_label}')

                # 检查组件
                elif any(detected_label in component for component in self.components_classes.values()):
                    classified_items['components'].append(detected_label)
                    print(f'Matched to component: {detected_label}')

                # 检查工具
                elif any(detected_label in tool for tool in self.tools_classes.values()):
                    classified_items['tools'].append(detected_label)
                    print(f'Matched to tool: {detected_label}')

                else:
                    print(f'Warning: No match found for {detected_label}')

        print(f"Classified items: {classified_items}")
        return classified_items

    def error_validation(self, classified, step_details, operator_name, location, item_type, task): # 检查分类后的物体是否存在错误，并生成错误日志
        details = {
            'now': datetime.now().strftime("%Y-%m-%d %H:%M"),
            'operator_name': self.operator_name,
            'location': location,
            'expected': step_details[item_type],
            'actual': classified[item_type],
            'step': step_details['step'],
            'task': task
        }

        error_result = {
            'type': item_type,
            'specific': details['actual'],
            'result': True
        }

        # 修改这里的比较逻辑
        expected_set = set(item.split(',')[0] for item in details['expected'].split(';'))
        actual_set = set(details['actual'])

        if expected_set.issubset(actual_set): # if actual_set.issubset(expected_set):
            error_result['result'] = True
            error_log = None
        else:
            error_result['result'] = False
            error_log = self.error_templates[item_type].format(**details)

            errorLog_dir = CONFIG['results_errorlog_dir']
            current_time = datetime.now().strftime("%Y-%m-%d_%H-%M-%S")
            errorLog_filename = f"{errorLog_dir}/text{current_time}.txt"
            with open(errorLog_filename, "w") as text_file:
                text_file.write(error_log)
            print(f"Error log saved.")

        return error_result, error_log

    def annotate_image_with_labels(self, image, detected_items, classified_items, item_type, error_result): # 根据错误情况来对实时图像中存在的所有物体进行标记
        # 注意：OpenCV 使用 BGR 颜色空间
        correct_color = (0, 255, 0)  # 绿色
        wrong_color = (0, 0, 255)    # 红色
        neutral_color = (128, 128, 128)  # 灰色

        processed_image = self.postprocess_image(image)
        if processed_image is None:
            print("Failed to process image for annotation")
            return None

        if detected_items is None or (isinstance(detected_items, np.ndarray) and detected_items.size == 0):
            print("No items detected for annotation")
            return processed_image

        print(f"Annotating for item_type: {item_type}")
        print(f"Classified items: {classified_items}")
        print(f"Error result: {error_result}")

        for detection in detected_items:
            x1, y1, x2, y2, conf, cls = detection[:6]
            detection_label = self.yolov7_label_order[int(cls)]
            print(f"Processing detection: {detection_label}")

            # 修改这里的逻辑
            if any(detection_label in item for item in classified_items[item_type]):
                if error_result['result']:
                    color = correct_color
                    label = detection_label
                else:
                    color = wrong_color
                    label = "Error" # 当有错误时，将标签改为"Error"
                    print(f" - In classified items, color: {color}")
            else:
                color = neutral_color
                label = detection_label
                print(f" - Not in classified items, color: {color}")

            cv2.rectangle(processed_image, (int(x1), int(y1)), (int(x2), int(y2)), color, 2)
            cv2.putText(processed_image, label, (int(x1), int(y1) - 10), cv2.FONT_HERSHEY_SIMPLEX, 0.5, color, 2)

        # 提高亮度和饱和度
        processed_image = self.enhance_image(processed_image)

        # 转换颜色空间从 BGR 到 RGB
        processed_image = cv2.cvtColor(processed_image, cv2.COLOR_BGR2RGB)

        timestamp = datetime.now().strftime("%Y%m%d%H%M%S")
        annotated_image_path = f'{CONFIG["results_image_dir"]}/annotated_{item_type}_{timestamp}.jpg'
        try:
            os.makedirs(os.path.dirname(annotated_image_path), exist_ok=True)
            # 注意：这里我们保存为BGR格式，因为cv2.imwrite期望BGR格式
            cv2_image = cv2.cvtColor(processed_image, cv2.COLOR_RGB2BGR)
            success = cv2.imwrite(annotated_image_path, cv2_image)
            if success:
                print(f"Annotated image saved to {annotated_image_path}")
            else:
                print(f"Failed to save annotated image: cv2.imwrite returned False")
        except Exception as e:
            print(f"Failed to save annotated image: {str(e)}")

        return processed_image

    def generate_prompt(self, step_details, error_description): # 获取将要传给GPT的prompt模板
        prompt_template = self.gpt_prompt_df['prompt'].iloc[0]
        prompt = prompt_template.format(step_details=step_details, error_description=error_description)
        return prompt

    def gpt_tts(self, prompt): # 利用GPT生成语音提醒，输出语音地址
        api_key = os.getenv('OPENAI_API_KEY')
        if not api_key:
            raise ValueError("API key is not set. Please ensure the 'OPENAI_API_KEY' environment variable is defined.")

        response = openai.chat.completions.create(
            model="gpt-4o",
            messages=[{"role": "user", "content": prompt}]
        )
        text = response.choices[0].message.content.strip()
        self.update_instruction_text(text)

        results_text_dir = CONFIG['results_text_dir']
        current_time = datetime.now().strftime("%Y-%m-%d_%H-%M-%S")
        text_filename = f"{results_text_dir}/text{current_time}.txt"
        with open(text_filename, "w") as text_file:
            text_file.write(text)
        print(f"Results text saved.")

        self.text_to_speech(text)


        '''
        print("GPT generated text:", text)  # 打印生成的文本
        try:
            self.update_instruction_text(text)
            print("GPT Text instruction updated")
        except Exception as e:
            print(f"Error updating text instruction: {e}")

        results_text_dir = CONFIG['results_text_dir']
        current_time = datetime.now().strftime("%Y-%m-%d_%H-%M-%S")
        text_filename = f"{results_text_dir}/text{current_time}.txt"
        with open(text_filename, "w") as text_file:
            text_file.write(text)
        print(f"Results text saved.")

        headers = {
            'Authorization': f'Bearer {api_key}',
            'Content-Type': 'application/json',
        }
        data = {
            "model": "tts-1",
            "input": text,
            "voice": CONFIG['tts_voice'],
            "speed": 0.8
        }
        response = requests.post('https://api.openai.com/v1/audio/speech', headers=headers, json=data)
        if response.status_code == 200:
            speech_filename = f"{CONFIG['results_speech_dir']}/speech{current_time}.mp3"
            with open(speech_filename, 'wb') as file:
                file.write(response.content)
            print("Error instruction speech saved.")
            return speech_filename
        else:
            print("Failed to generate speech:", response.status_code, response.text)
            return None
        '''

    def text_to_speech(self, text): # 把除了GPT以外的文字转换成语音，输出语音地址
        timestamp = datetime.now().strftime("%Y%m%d%H%M%S")
        voice_path = f'{CONFIG["TTS_speech_dir"]}/voice_{timestamp}.mp3'
        try:
            engine = pyttsx3.init()
            rate = engine.getProperty('rate')
            engine.setProperty('rate', rate - 80)
            volume = engine.getProperty('volume')
            engine.setProperty('volume', volume + 0.25)
            voices = engine.getProperty('voices')
            engine.setProperty('voice', voices[1].id)
            engine.say(text)
            engine.save_to_file(text, voice_path)
            engine.runAndWait()
            self.current_audio_file = voice_path
            return voice_path
        except Exception as e:
            print(f"Error with text-to-speech: {e}")
            return None

    def get_step_details(self, index): # 从预先加载的装配任务数据中提取特定步骤的详细信息。
        self.steps_classes = self.assembly_tasks_df['step'].dropna().to_dict()
        self.components_classes = self.assembly_tasks_df['components'].dropna().to_dict()
        self.tools_classes = self.assembly_tasks_df['tools'].dropna().to_dict()
        self.operations_classes = self.assembly_tasks_df['operations'].dropna().to_dict()
        self.time_classes = self.assembly_tasks_df['time'].dropna().to_dict()
        self.lastorder_classes = self.assembly_tasks_df['lastorder'].dropna().to_dict()
        return {
            'components': self.components_classes[index],
            'tools': self.tools_classes[index],
            'operations': self.operations_classes[index],
            'time': self.time_classes[index],
            'step': self.steps_classes[index],
            'steps': self.steps_classes[index]
        }

    def process_step(self, index, item_type, step_details): # 装配步骤的推进
        self.progress_text.delete('1.0', tk.END)
        text = f"Start assembly step{index+1}.{item_type}."
        self.update_progress_text(text + "\n")

        if step_details[item_type] != "None":
            retry = True
            retry_count = 0
            while retry and retry_count < 3:
                success = self.handle_step(index, item_type, step_details)
                if not success:
                    if retry_count < 2:
                        self.handle_error(index, item_type, step_details)
                        retry_count += 1
                    else:
                        self.update_progress_text("\nFailed to correct the error after 2 attempts.\n")
                        retry = False
                else:
                    success_text = "\nYou did it correctly!\n"
                    self.update_progress_text(success_text)
                    voice_path = self.text_to_speech(success_text)
                    if voice_path:
                        self.play_audio(voice_path)
                    self.update_progress_text(f"\nEnd step{index+1}.{item_type}\n")
                    retry = False

        self.window.update()

    def handle_step(self, index, item_type, step_details): # 区分操作类型，然后开展细分任务
        self.error_result = {'result': True}

        if self.error_result['result']:  # 只有在没有发生错误的情况下才播放原始指示
            if item_type in ['components', 'tools']:
                task = f"Please prepare the following {item_type}: {step_details[item_type]}."
                sleep_time = 0.5 # 设置抓取零件和工具的时间
            else:
                task = f"Please follow the instructions to complete the step: {step_details['operations']}."
                sleep_time = 1
                # sleep_time = step_details['time'] # 按照每个装配步骤原定的时长来设置时间

            self.update_instruction_text(task)
            self.window.update()
            time.sleep(0.1)

            voice_path = self.text_to_speech(task)
            if voice_path:
                self.play_audio(voice_path)
            else:
                print("Failed to generate speech for task")

            time.sleep(sleep_time)

        image = self.capture_image()
        if image is not None:
            self.update_realtime_image(image)
            self.window.update()
            time.sleep(0.1)

            preprocessed_image = self.preprocess_image(image)
            if preprocessed_image is not None:
                detected_items = self.detect_items(preprocessed_image)
                if detected_items is not None and len(detected_items) > 0:
                    classified_items = self.classify_detections(detected_items)

                    text = "\nDetected items:\n"
                    for det in detected_items:
                        x1, y1, x2, y2, conf, cls = det[:6]  # 获取坐标和类别信息
                        label = self.yolov7_label_order[int(cls)]
                        text += f"{label} (confidence: {conf:.2f}.)\n"
                    self.update_progress_text(text)
                    self.window.update()
                    time.sleep(0.1)

                    self.error_result, self.error_log = self.error_validation(
                        classified_items, step_details, self.operator_name, 'location', item_type, task
                    )

                    text = f"\nError Log: {self.error_log}."
                    self.update_progress_text(text)
                    self.window.update()
                    time.sleep(0.1)

                    annotated_image = self.annotate_image_with_labels(
                        image, detected_items, classified_items, item_type, self.error_result
                    )
                    if annotated_image is not None:
                        self.update_realtime_image(annotated_image)
                    else:
                        print("Failed to annotate image")
                    self.window.update()
                    time.sleep(0.1)
                else:
                    print("No items detected or detection failed")
                    self.update_progress_text("No items detected or detection failed.\n")
            else:
                print("Failed to preprocess image")
                self.update_progress_text("Failed to preprocess image.\n")
        else:
            print("Failed to capture image")
            self.update_progress_text("Failed to capture image.\n")

        self.window.update()
        time.sleep(0.1)  # 给GUI一些时间来刷新

        return self.error_result.get('result', False)

    def handle_error(self, index, item_type, step_details): # 装配流程中的错误处理
        prompt = self.generate_prompt(step_details, self.error_log)
        speech_filename = self.gpt_tts(prompt)
        if speech_filename:
            self.play_audio(speech_filename)
        self.play_audio(speech_filename)
        text = f"\nRedo step{index+1}.{item_type}"
        self.update_progress_text(text)
        self.window.update()

    def on_closing(self): # 在主窗口关闭时停止所有正在播放的音频
        pygame.mixer.music.stop()
        pygame.mixer.quit()
        self.window.destroy()

    def run(self):
        print("Starting the Assembly Monitoring System...")
        try:
            for index in range(2):
            # 本来想要循环数据表中的所有步骤，但现在先只做前两个步骤
            # for index in range(self.assembly_tasks_df.dropna(how='all').shape[0] - 1):
                step_details = self.get_step_details(index)
                step_number = int(''.join(filter(str.isdigit, step_details['step'])))
                self.update_gui_4image(step_number)
                self.progress_text.delete('1.0', tk.END)
                self.window.update()
                time.sleep(0.1)

                for item_type in ['components', 'tools', 'steps']:
                    self.process_step(index, item_type, step_details)
                    self.window.update()

            completion_message = "All assembly tasks have been successfully completed!"
            self.progress_text.delete('1.0', tk.END)
            self.update_progress_text("\n" + completion_message + "\n")

            voice_path = self.text_to_speech(completion_message)
            if voice_path:
                self.play_audio(voice_path)

            self.window.update()

        except Exception as e:
            print(f"An error occurred during execution: {e}")
            import traceback
            traceback.print_exc()
        finally:
            print("Assembly Monitoring System has finished running.")

if __name__ == '__main__':
    root = tk.Tk()
    app = AssemblyMonitoringSystem(root)
    time.sleep(2)
    app.run()
    root.mainloop()
